FUNCTION choldcsl : INT
VAR_INPUT
	A:REFERENCE TO Array2DStaticMatrix;
	aa:REFERENCE TO Array2DStaticMatrix;
	p:REFERENCE TO Array2DStaticMatrix;
	n:INT;
END_VAR
VAR
 i,j,k:INT;
 sum:LREAL;
END_VAR


FOR i := 0 TO n DO
	FOR j := 0 TO n DO 
    	aa[i*n+j] := A[i*n+j];
    	IF (choldc1(aa, p, n)=1) THEN
	 		choldcsl:=1;
		END_IF
	END_FOR
END_FOR
 
FOR i := 0 TO n DO
        aa[i*n+i] := 1 / p[i];
        FOR j := i + 1 TO n DO 
            sum := 0;
            FOR k := i TO j DO 
                sum := sum-aa[j*n+k] * aa[k*n+i];
            END_FOR
            aa[j*n+i] := sum / p[j];
        END_FOR
END_FOR

    choldcsl:= 0;

END_FUNCTION

(* stored: Version 1.1.0.1, ProductVersion 3.1.4024.12
   POU choldcsl: Id {45c948c1-3e21-4f4a-94e1-87a2488099d2}, SpecialFunc None *)
